LIN {X 0,Y 228.943,Z 711.605,A -85,B 0,C 180,E1 6110.84,E2 6110.84} C_VEL
LIN {X 0,Y 224.559,Z 717.902,A -85,B 0,C 180,E1 6110.576,E2 6110.576} C_VEL
LIN {X 0,Y 211.936,Z 735.349,A -85,B 0,C 180,E1 6108.891,E2 6108.891} C_VEL
LIN {X 0,Y 198.221,Z 751.661,A -85,B 0,C 180,E1 6106.779,E2 6106.779} C_VEL
LIN {X 0,Y 183.955,Z 766.558,A -85,B 0,C 180,E1 6104.16,E2 6104.16} C_VEL
LIN {X 0,Y 168.446,Z 780.857,A -85,B 0,C 180,E1 6100.693,E2 6100.693} C_VEL
LIN {X 0,Y 153.69,Z 792.992,A -85,B 0,C 180,E1 6096.531,E2 6096.531} C_VEL
LIN {X 0,Y 138.441,Z 804.254,A -85,B 0,C 180,E1 6090.912,E2 6090.912} C_VEL
LIN {X 0,Y 124.785,Z 813.422,A -85,B 0,C 180,E1 6084.023,E2 6084.023} C_VEL
LIN {X 0,Y 112.729,Z 821.12,A -85,B 0,C 180,E1 6075.198,E2 6075.198} C_VEL
LIN {X 0,Y 103.673,Z 826.988,A -85,B 0,C 180,E1 6064.681,E2 6064.681} C_VEL
LIN {X 0,Y 98.168,Z 831.113,A -85,B 0,C 180,E1 6052.77,E2 6052.77} C_VEL
LIN {X 0,Y 96.317,Z 833.266,A -85,B 0,C 180,E1 6041.375,E2 6041.375} C_VEL
LIN {X 0,Y 96.353,Z 833.983,A -85,B 0,C 180,E1 6032.974,E2 6032.974} C_VEL
LIN {X 0,Y 96.353,Z 833.978,A -85,B 0,C 180,E1 6027.026,E2 6027.026} C_VEL
LIN {X 0,Y 96.32,Z 833.25,A -85,B 0,C 180,E1 6018.625,E2 6018.625} C_VEL
LIN {X 0,Y 98.345,Z 830.901,A -85,B 0,C 180,E1 6006.641,E2 6006.641} C_VEL
LIN {X 0,Y 104.029,Z 826.718,A -85,B 0,C 180,E1 5994.78,E2 5994.78} C_VEL
LIN {X 0,Y 113.237,Z 820.733,A -85,B 0,C 180,E1 5984.341,E2 5984.341} C_VEL
LIN {X 0,Y 125.437,Z 812.892,A -85,B 0,C 180,E1 5975.582,E2 5975.582} C_VEL
LIN {X 0,Y 139.162,Z 803.604,A -85,B 0,C 180,E1 5968.774,E2 5968.774} C_VEL
LIN {X 0,Y 154.481,Z 792.265,A -85,B 0,C 180,E1 5963.212,E2 5963.212} C_VEL
LIN {X 0,Y 170.131,Z 779.252,A -85,B 0,C 180,E1 5958.885,E2 5958.885} C_VEL
LIN {X 0,Y 184.827,Z 765.494,A -85,B 0,C 180,E1 5955.656,E2 5955.656} C_VEL
LIN {X 0,Y 199.569,Z 749.867,A -85,B 0,C 180,E1 5952.984,E2 5952.984} C_VEL
LIN {X 0,Y 212.851,Z 733.839,A -85,B 0,C 180,E1 5950.966,E2 5950.966} C_VEL
LIN {X 0,Y 225.524,Z 716.172,A -85,B 0,C 180,E1 5949.294,E2 5949.294} C_VEL
LIN {X 0,Y 236.712,Z 697.903,A -85,B 0,C 180,E1 5947.997,E2 5947.997} C_VEL
LIN {X 0,Y 246.77,Z 678.537,A -85,B 0,C 180,E1 5946.946,E2 5946.946} C_VEL
LIN {X 0,Y 255.417,Z 658.457,A -85,B 0,C 180,E1 5946.129,E2 5946.129} C_VEL
LIN {X 0,Y 262.423,Z 638.201,A -85,B 0,C 180,E1 5945.52,E2 5945.52} C_VEL
LIN {X 0,Y 267.944,Z 616.978,A -85,B 0,C 180,E1 5945.047,E2 5945.047} C_VEL
LIN {X 0,Y 271.895,Z 594.865,A -85,B 0,C 180,E1 5944.639,E2 5944.639} C_VEL
LIN {X 0,Y 282.099,Z 508.002,A -85,B 0,C 180,E1 5943.2,E2 5943.2} C_VEL
LIN {X 0,Y 281.259,Z 505.176,A -85,B 0,C 180,E1 5939.389,E2 5939.389} C_VEL
LIN {X 0,Y 281.202,Z 505.463,A -85,B 0,C 180,E1 5936.126,E2 5936.126} C_VEL
LIN {X 0,Y 281.88,Z 508.582,A -85,B 0,C 180,E1 5932.471,E2 5932.471} C_VEL
LIN {X 0,Y 271.081,Z 600.166,A -85,B 0,C 180,E1 5931.031,E2 5931.031} C_VEL
LIN {X 0,Y 266.657,Z 621.932,A -85,B 0,C 180,E1 5930.606,E2 5930.606} C_VEL
LIN {X 0,Y 260.873,Z 642.254,A -85,B 0,C 180,E1 5930.059,E2 5930.059} C_VEL
LIN {X 0,Y 253.227,Z 663.066,A -85,B 0,C 180,E1 5929.305,E2 5929.305} C_VEL
LIN {X 0,Y 244.471,Z 682.335,A -85,B 0,C 180,E1 5928.379,E2 5928.379} C_VEL
LIN {X 0,Y 234.272,Z 700.902,A -85,B 0,C 180,E1 5927.212,E2 5927.212} C_VEL
LIN {X 0,Y 223.26,Z 717.863,A -85,B 0,C 180,E1 5925.826,E2 5925.826} C_VEL
LIN {X 0,Y 210.147,Z 735.251,A -85,B 0,C 180,E1 5923.96,E2 5923.96} C_VEL
LIN {X 0,Y 196.844,Z 750.52,A -85,B 0,C 180,E1 5921.774,E2 5921.774} C_VEL
LIN {X 0,Y 182.156,Z 765.197,A -85,B 0,C 180,E1 5918.924,E2 5918.924} C_VEL
LIN {X 0,Y 167.162,Z 778.201,A -85,B 0,C 180,E1 5915.388,E2 5915.388} C_VEL
LIN {X 0,Y 152.898,Z 789.101,A -85,B 0,C 180,E1 5911.194,E2 5911.194} C_VEL
LIN {X 0,Y 138.176,Z 799.134,A -85,B 0,C 180,E1 5905.578,E2 5905.578} C_VEL
LIN {X 0,Y 124.994,Z 807.232,A -85,B 0,C 180,E1 5898.756,E2 5898.756} C_VEL
LIN {X 0,Y 113.323,Z 813.809,A -85,B 0,C 180,E1 5890.096,E2 5890.096} C_VEL
LIN {X 0,Y 104.467,Z 818.511,A -85,B 0,C 180,E1 5879.847,E2 5879.847} C_VEL
LIN {X 0,Y 98.88,Z 821.593,A -85,B 0,C 180,E1 5868.097,E2 5868.097} C_VEL
LIN {X 0,Y 96.719,Z 823.052,A -85,B 0,C 180,E1 5856.529,E2 5856.529} C_VEL
LIN {X 0,Y 96.52,Z 823.179,A -85,B 0,C 180,E1 5847.031,E2 5847.031} C_VEL
LIN {X 0,Y 97.582,Z 822.439,A -85,B 0,C 180,E1 5836.973,E2 5836.973} C_VEL
LIN {X 0,Y 101.63,Z 820.074,A -85,B 0,C 180,E1 5824.974,E2 5824.974} C_VEL
LIN {X 0,Y 109.093,Z 816.103,A -85,B 0,C 180,E1 5814.087,E2 5814.087} C_VEL
LIN {X 0,Y 119.622,Z 810.413,A -85,B 0,C 180,E1 5804.728,E2 5804.728} C_VEL
LIN {X 0,Y 132.62,Z 802.775,A -85,B 0,C 180,E1 5796.952,E2 5796.952} C_VEL
LIN {X 0,Y 146.033,Z 794.058,A -85,B 0,C 180,E1 5791.149,E2 5791.149} C_VEL
LIN {X 0,Y 161.435,Z 782.868,A -85,B 0,C 180,E1 5786.098,E2 5786.098} C_VEL
LIN {X 0,Y 176.171,Z 770.745,A -85,B 0,C 180,E1 5782.32,E2 5782.32} C_VEL
LIN {X 0,Y 190.669,Z 757.19,A -85,B 0,C 180,E1 5779.286,E2 5779.286} C_VEL
LIN {X 0,Y 204.72,Z 742.023,A -85,B 0,C 180,E1 5776.815,E2 5776.815} C_VEL
LIN {X 0,Y 217.286,Z 726.43,A -85,B 0,C 180,E1 5774.916,E2 5774.916} C_VEL
LIN {X 0,Y 229.6,Z 708.754,A -85,B 0,C 180,E1 5773.278,E2 5773.278} C_VEL
LIN {X 0,Y 240.308,Z 690.764,A -85,B 0,C 180,E1 5772.008,E2 5772.008} C_VEL
LIN {X 0,Y 249.916,Z 671.405,A -85,B 0,C 180,E1 5770.959,E2 5770.959} C_VEL
LIN {X 0,Y 257.672,Z 652.265,A -85,B 0,C 180,E1 5770.173,E2 5770.173} C_VEL
LIN {X 0,Y 264.628,Z 630.575,A -85,B 0,C 180,E1 5769.505,E2 5769.505} C_VEL
LIN {X 0,Y 269.675,Z 609.251,A -85,B 0,C 180,E1 5769.034,E2 5769.034} C_VEL
LIN {X 0,Y 273.096,Z 587.225,A -85,B 0,C 180,E1 5768.661,E2 5768.661} C_VEL
LIN {X 0,Y 282.119,Z 508.77,A -85,B 0,C 180,E1 5767.415,E2 5767.415} C_VEL
LIN {X 0,Y 281.448,Z 505.359,A -85,B 0,C 180,E1 5763.259,E2 5763.259} C_VEL
LIN {X 0,Y 281.564,Z 505.603,A -85,B 0,C 180,E1 5760.204,E2 5760.204} C_VEL
LIN {X 0,Y 282.328,Z 508.47,A -85,B 0,C 180,E1 5756.755,E2 5756.755} C_VEL
LIN {X 0,Y 271.257,Z 601.222,A -85,B 0,C 180,E1 5755.259,E2 5755.259} C_VEL
LIN {X 0,Y 266.713,Z 623.38,A -85,B 0,C 180,E1 5754.832,E2 5754.832} C_VEL
LIN {X 0,Y 260.73,Z 644.157,A -85,B 0,C 180,E1 5754.332,E2 5754.332} C_VEL
LIN {X 0,Y 252.828,Z 665.462,A -85,B 0,C 180,E1 5753.624,E2 5753.624} C_VEL
LIN {X 0,Y 243.909,Z 684.958,A -85,B 0,C 180,E1 5752.749,E2 5752.749} C_VEL
LIN {X 0,Y 233.45,Z 703.978,A -85,B 0,C 180,E1 5751.625,E2 5751.625} C_VEL
LIN {X 0,Y 224.559,Z 717.902,A -85,B 0,C 180,E1 5750.576,E2 5750.576} C_VEL
LIN {X 0,Y 220.012,Z 724.207,A -85,B 0,C 180,E1 5750.279,E2 5750.279} C_VEL
LIN {X 0,Y 206.999,Z 739.459,A -85,B 0,C 180,E1 5750.323,E2 5750.323} C_VEL
LIN {X 0,Y 201.901,Z 745.116,A -85,B 0,C 180,E1 5749.921,E2 5749.921} C_VEL
LIN {X 0,Y 187.314,Z 760.779,A -85,B 0,C 180,E1 5747.635,E2 5747.635} C_VEL
LIN {X 0,Y 172.824,Z 774.387,A -85,B 0,C 180,E1 5744.91,E2 5744.91} C_VEL
LIN {X 0,Y 156.438,Z 787.999,A -85,B 0,C 180,E1 5741.068,E2 5741.068} C_VEL
LIN {X 0,Y 140.822,Z 799.498,A -85,B 0,C 180,E1 5736.333,E2 5736.333} C_VEL
LIN {X 0,Y 125.674,Z 809.548,A -85,B 0,C 180,E1 5730.132,E2 5730.132} C_VEL
LIN {X 0,Y 111.697,Z 817.971,A -85,B 0,C 180,E1 5721.973,E2 5721.973} C_VEL
LIN {X 0,Y 100.404,Z 824.489,A -85,B 0,C 180,E1 5711.85,E2 5711.85} C_VEL
LIN {X 0,Y 92.315,Z 829.427,A -85,B 0,C 180,E1 5699.168,E2 5699.168} C_VEL
LIN {X 0,Y 88.754,Z 832.327,A -85,B 0,C 180,E1 5686.358,E2 5686.358} C_VEL
LIN {X 0,Y 88.313,Z 833.461,A -85,B 0,C 180,E1 5674.936,E2 5674.936} C_VEL
LIN {X 0,Y 88.388,Z 833.582,A -85,B 0,C 180,E1 5668.055,E2 5668.055} C_VEL
LIN {X 0,Y 88.311,Z 832.952,A -85,B 0,C 180,E1 5658.903,E2 5658.903} C_VEL
LIN {X 0,Y 90.258,Z 830.908,A -85,B 0,C 180,E1 5646.498,E2 5646.498} C_VEL
LIN {X 0,Y 96.203,Z 826.924,A -85,B 0,C 180,E1 5633.673,E2 5633.673} C_VEL
LIN {X 0,Y 106.474,Z 820.908,A -85,B 0,C 180,E1 5622.111,E2 5622.111} C_VEL
LIN {X 0,Y 118.725,Z 813.708,A -85,B 0,C 180,E1 5613.517,E2 5613.517} C_VEL
LIN {X 0,Y 133.055,Z 804.664,A -85,B 0,C 180,E1 5606.593,E2 5606.593} C_VEL
LIN {X 0,Y 148.088,Z 794.164,A -85,B 0,C 180,E1 5601.296,E2 5601.296} C_VEL
LIN {X 0,Y 164.141,Z 781.647,A -85,B 0,C 180,E1 5596.995,E2 5596.995} C_VEL
LIN {X 0,Y 179.162,Z 768.454,A -85,B 0,C 180,E1 5593.827,E2 5593.827} C_VEL
LIN {X 0,Y 194.185,Z 753.452,A -85,B 0,C 180,E1 5591.229,E2 5591.229} C_VEL
LIN {X 0,Y 207.964,Z 737.594,A -85,B 0,C 180,E1 5589.235,E2 5589.235} C_VEL
LIN {X 0,Y 220.914,Z 720.48,A -85,B 0,C 180,E1 5587.62,E2 5587.62} C_VEL
LIN {X 0,Y 232.396,Z 702.941,A -85,B 0,C 180,E1 5586.37,E2 5586.37} C_VEL
LIN {X 0,Y 243.011,Z 683.835,A -85,B 0,C 180,E1 5585.334,E2 5585.334} C_VEL
LIN {X 0,Y 251.753,Z 664.803,A -85,B 0,C 180,E1 5584.555,E2 5584.555} C_VEL
LIN {X 0,Y 259.563,Z 643.938,A -85,B 0,C 180,E1 5583.918,E2 5583.918} C_VEL
LIN {X 0,Y 265.684,Z 622.813,A -85,B 0,C 180,E1 5583.45,E2 5583.45} C_VEL
LIN {X 0,Y 270.213,Z 600.861,A -85,B 0,C 180,E1 5583.054,E2 5583.054} C_VEL
LIN {X 0,Y 280.622,Z 514.878,A -85,B 0,C 180,E1 5581.689,E2 5581.689} C_VEL
LIN {X 0,Y 280.248,Z 513.095,A -85,B 0,C 180,E1 5579.182,E2 5579.182} C_VEL
LIN {X 0,Y 280.208,Z 513.353,A -85,B 0,C 180,E1 5576.317,E2 5576.317} C_VEL
LIN {X 0,Y 280.468,Z 515.368,A -85,B 0,C 180,E1 5573.991,E2 5573.991} C_VEL
LIN {X 0,Y 270.229,Z 600.323,A -85,B 0,C 180,E1 5572.716,E2 5572.716} C_VEL
LIN {X 0,Y 265.751,Z 622.044,A -85,B 0,C 180,E1 5572.319,E2 5572.319} C_VEL
LIN {X 0,Y 259.977,Z 642.117,A -85,B 0,C 180,E1 5571.819,E2 5571.819} C_VEL
LIN {X 0,Y 252.47,Z 662.437,A -85,B 0,C 180,E1 5571.14,E2 5571.14} C_VEL
LIN {X 0,Y 244.087,Z 680.892,A -85,B 0,C 180,E1 5570.331,E2 5570.331} C_VEL
LIN {X 0,Y 234.04,Z 699.126,A -85,B 0,C 180,E1 5569.288,E2 5569.288} C_VEL
LIN {X 0,Y 222.222,Z 717.316,A -85,B 0,C 180,E1 5567.932,E2 5567.932} C_VEL
LIN {X 0,Y 209.447,Z 734.138,A -85,B 0,C 180,E1 5566.274,E2 5566.274} C_VEL
LIN {X 0,Y 196.278,Z 749.177,A -85,B 0,C 180,E1 5564.314,E2 5564.314} C_VEL
LIN {X 0,Y 182.04,Z 763.217,A -85,B 0,C 180,E1 5561.838,E2 5561.838} C_VEL
LIN {X 0,Y 167.34,Z 775.94,A -85,B 0,C 180,E1 5558.761,E2 5558.761} C_VEL
LIN {X 0,Y 152.39,Z 787.337,A -85,B 0,C 180,E1 5554.879,E2 5554.879} C_VEL
LIN {X 0,Y 137.245,Z 797.507,A -85,B 0,C 180,E1 5549.822,E2 5549.822} C_VEL
LIN {X 0,Y 122.453,Z 806.219,A -85,B 0,C 180,E1 5543.147,E2 5543.147} C_VEL
LIN {X 0,Y 110.002,Z 812.815,A -85,B 0,C 180,E1 5535.15,E2 5535.15} C_VEL
LIN {X 0,Y 99.13,Z 818.185,A -85,B 0,C 180,E1 5524.39,E2 5524.39} C_VEL
LIN {X 0,Y 92.208,Z 821.597,A -85,B 0,C 180,E1 5512.304,E2 5512.304} C_VEL
LIN {X 0,Y 89.124,Z 823.234,A -85,B 0,C 180,E1 5500.34,E2 5500.34} C_VEL
LIN {X 0,Y 88.502,Z 823.711,A -85,B 0,C 180,E1 5489.353,E2 5489.353} C_VEL
LIN {X 0,Y 89.302,Z 823.135,A -85,B 0,C 180,E1 5478.374,E2 5478.374} C_VEL
LIN {X 0,Y 92.936,Z 821.275,A -85,B 0,C 180,E1 5465.87,E2 5465.87} C_VEL
LIN {X 0,Y 100.36,Z 817.677,A -85,B 0,C 180,E1 5454,E2 5454} C_VEL
LIN {X 0,Y 111.086,Z 812.343,A -85,B 0,C 180,E1 5443.942,E2 5443.942} C_VEL
LIN {X 0,Y 124.421,Z 805.188,A -85,B 0,C 180,E1 5435.745,E2 5435.745} C_VEL
LIN {X 0,Y 138.94,Z 796.519,A -85,B 0,C 180,E1 5429.456,E2 5429.456} C_VEL
LIN {X 0,Y 154.245,Z 786.199,A -85,B 0,C 180,E1 5424.512,E2 5424.512} C_VEL
LIN {X 0,Y 169.828,Z 774.115,A -85,B 0,C 180,E1 5420.597,E2 5420.597} C_VEL
LIN {X 0,Y 184.615,Z 761.006,A -85,B 0,C 180,E1 5417.603,E2 5417.603} C_VEL
LIN {X 0,Y 199.384,Z 745.999,A -85,B 0,C 180,E1 5415.116,E2 5415.116} C_VEL
LIN {X 0,Y 212.601,Z 730.569,A -85,B 0,C 180,E1 5413.222,E2 5413.222} C_VEL
LIN {X 0,Y 225.009,Z 713.713,A -85,B 0,C 180,E1 5411.659,E2 5411.659} C_VEL
LIN {X 0,Y 235.864,Z 696.432,A -85,B 0,C 180,E1 5410.439,E2 5410.439} C_VEL
LIN {X 0,Y 246.247,Z 676.879,A -85,B 0,C 180,E1 5409.374,E2 5409.374} C_VEL
LIN {X 0,Y 254.801,Z 657.342,A -85,B 0,C 180,E1 5408.569,E2 5408.569} C_VEL
LIN {X 0,Y 261.963,Z 636.81,A -85,B 0,C 180,E1 5407.933,E2 5407.933} C_VEL
LIN {X 0,Y 267.47,Z 615.741,A -85,B 0,C 180,E1 5407.456,E2 5407.456} C_VEL
LIN {X 0,Y 271.403,Z 593.852,A -85,B 0,C 180,E1 5407.088,E2 5407.088} C_VEL
LIN {X 0,Y 280.729,Z 515.352,A -85,B 0,C 180,E1 5405.878,E2 5405.878} C_VEL
LIN {X 0,Y 280.444,Z 513.234,A -85,B 0,C 180,E1 5402.657,E2 5402.657} C_VEL
LIN {X 0,Y 280.552,Z 513.477,A -85,B 0,C 180,E1 5400.409,E2 5400.409} C_VEL
LIN {X 0,Y 280.864,Z 515.249,A -85,B 0,C 180,E1 5398.276,E2 5398.276} C_VEL
LIN {X 0,Y 270.432,Z 601.099,A -85,B 0,C 180,E1 5396.948,E2 5396.948} C_VEL
LIN {X 0,Y 265.812,Z 623.347,A -85,B 0,C 180,E1 5396.547,E2 5396.547} C_VEL
LIN {X 0,Y 259.811,Z 643.945,A -85,B 0,C 180,E1 5396.09,E2 5396.09} C_VEL
LIN {X 0,Y 251.756,Z 665.383,A -85,B 0,C 180,E1 5395.434,E2 5395.434} C_VEL
LIN {X 0,Y 243.015,Z 684.289,A -85,B 0,C 180,E1 5394.655,E2 5394.655} C_VEL
LIN {X 0,Y 232.401,Z 703.346,A -85,B 0,C 180,E1 5393.619,E2 5393.619} C_VEL
LIN {X 0,Y 220.919,Z 720.814,A -85,B 0,C 180,E1 5392.369,E2 5392.369} C_VEL
LIN {X 0,Y 207.215,Z 738.779,A -85,B 0,C 180,E1 5390.655,E2 5390.655} C_VEL
LIN {X 0,Y 201.901,Z 745.116,A -85,B 0,C 180,E1 5389.921,E2 5389.921} C_VEL
LIN {X 0,Y 196.629,Z 750.729,A -85,B 0,C 180,E1 5389.468,E2 5389.468} C_VEL
LIN {X 0,Y 181.804,Z 764.258,A -85,B 0,C 180,E1 5389.155,E2 5389.155} C_VEL
LIN {X 0,Y 176.236,Z 769.222,A -85,B 0,C 180,E1 5388.563,E2 5388.563} C_VEL
LIN {X 0,Y 160.13,Z 782.767,A -85,B 0,C 180,E1 5385.42,E2 5385.42} C_VEL
LIN {X 0,Y 143.84,Z 794.82,A -85,B 0,C 180,E1 5381.353,E2 5381.353} C_VEL
LIN {X 0,Y 127.163,Z 805.736,A -85,B 0,C 180,E1 5375.792,E2 5375.792} C_VEL
LIN {X 0,Y 112.21,Z 814.524,A -85,B 0,C 180,E1 5368.803,E2 5368.803} C_VEL
LIN {X 0,Y 98.734,Z 821.792,A -85,B 0,C 180,E1 5359.419,E2 5359.419} C_VEL
LIN {X 0,Y 88.422,Z 827.177,A -85,B 0,C 180,E1 5347.633,E2 5347.633} C_VEL
LIN {X 0,Y 82.171,Z 830.859,A -85,B 0,C 180,E1 5333.674,E2 5333.674} C_VEL
LIN {X 0,Y 80.288,Z 832.717,A -85,B 0,C 180,E1 5320.329,E2 5320.329} C_VEL
LIN {X 0,Y 80.426,Z 833.189,A -85,B 0,C 180,E1 5310.712,E2 5310.712} C_VEL
LIN {X 0,Y 80.269,Z 832.903,A -85,B 0,C 180,E1 5302.125,E2 5302.125} C_VEL
LIN {X 0,Y 81.64,Z 831.213,A -85,B 0,C 180,E1 5288.444,E2 5288.444} C_VEL
LIN {X 0,Y 87.022,Z 827.945,A -85,B 0,C 180,E1 5274.662,E2 5274.662} C_VEL
LIN {X 0,Y 96.492,Z 822.877,A -85,B 0,C 180,E1 5262.635,E2 5262.635} C_VEL
LIN {X 0,Y 108.76,Z 816.303,A -85,B 0,C 180,E1 5253.221,E2 5253.221} C_VEL
LIN {X 0,Y 123.263,Z 808.018,A -85,B 0,C 180,E1 5245.795,E2 5245.795} C_VEL
LIN {X 0,Y 139.357,Z 797.829,A -85,B 0,C 180,E1 5239.97,E2 5239.97} C_VEL
LIN {X 0,Y 155.694,Z 786.056,A -85,B 0,C 180,E1 5235.579,E2 5235.579} C_VEL
LIN {X 0,Y 170.945,Z 773.62,A -85,B 0,C 180,E1 5232.378,E2 5232.378} C_VEL
LIN {X 0,Y 185.715,Z 760.038,A -85,B 0,C 180,E1 5229.865,E2 5229.865} C_VEL
LIN {X 0,Y 200.792,Z 744.156,A -85,B 0,C 180,E1 5227.733,E2 5227.733} C_VEL
LIN {X 0,Y 214.187,Z 727.761,A -85,B 0,C 180,E1 5226.127,E2 5226.127} C_VEL
LIN {X 0,Y 226.921,Z 709.717,A -85,B 0,C 180,E1 5224.802,E2 5224.802} C_VEL
LIN {X 0,Y 237.98,Z 691.361,A -85,B 0,C 180,E1 5223.789,E2 5223.789} C_VEL
LIN {X 0,Y 247.792,Z 671.982,A -85,B 0,C 180,E1 5222.974,E2 5222.974} C_VEL
LIN {X 0,Y 256.17,Z 651.514,A -85,B 0,C 180,E1 5222.337,E2 5222.337} C_VEL
LIN {X 0,Y 262.969,Z 630.411,A -85,B 0,C 180,E1 5221.863,E2 5221.863} C_VEL
LIN {X 0,Y 268.333,Z 607.61,A -85,B 0,C 180,E1 5221.467,E2 5221.467} C_VEL
LIN {X 0,Y 271.894,Z 583.958,A -85,B 0,C 180,E1 5221.1,E2 5221.1} C_VEL
LIN {X 0,Y 279.349,Z 521.673,A -85,B 0,C 180,E1 5220.153,E2 5220.153} C_VEL
LIN {X 0,Y 279.221,Z 520.995,A -85,B 0,C 180,E1 5218.768,E2 5218.768} C_VEL
LIN {X 0,Y 279.217,Z 521.278,A -85,B 0,C 180,E1 5216.467,E2 5216.467} C_VEL
LIN {X 0,Y 279.239,Z 522.27,A -85,B 0,C 180,E1 5215.53,E2 5215.53} C_VEL
LIN {X 0,Y 269.581,Z 600.652,A -85,B 0,C 180,E1 5214.408,E2 5214.408} C_VEL
LIN {X 0,Y 265.02,Z 622.436,A -85,B 0,C 180,E1 5214.038,E2 5214.038} C_VEL
LIN {X 0,Y 259.173,Z 642.455,A -85,B 0,C 180,E1 5213.576,E2 5213.576} C_VEL
LIN {X 0,Y 251.366,Z 663.216,A -85,B 0,C 180,E1 5212.934,E2 5212.934} C_VEL
LIN {X 0,Y 242.722,Z 681.885,A -85,B 0,C 180,E1 5212.172,E2 5212.172} C_VEL
LIN {X 0,Y 231.736,Z 701.355,A -85,B 0,C 180,E1 5211.125,E2 5211.125} C_VEL
LIN {X 0,Y 219.887,Z 719.001,A -85,B 0,C 180,E1 5209.876,E2 5209.876} C_VEL
LIN {X 0,Y 206.289,Z 736.307,A -85,B 0,C 180,E1 5208.249,E2 5208.249} C_VEL
LIN {X 0,Y 192.419,Z 751.52,A -85,B 0,C 180,E1 5206.329,E2 5206.329} C_VEL
LIN {X 0,Y 177.894,Z 765.368,A -85,B 0,C 180,E1 5203.963,E2 5203.963} C_VEL
LIN {X 0,Y 162.838,Z 777.788,A -85,B 0,C 180,E1 5201.008,E2 5201.008} C_VEL
LIN {X 0,Y 146.622,Z 789.48,A -85,B 0,C 180,E1 5197.011,E2 5197.011} C_VEL
LIN {X 0,Y 131.261,Z 799.17,A -85,B 0,C 180,E1 5192.078,E2 5192.078} C_VEL
LIN {X 0,Y 116.349,Z 807.457,A -85,B 0,C 180,E1 5185.585,E2 5185.585} C_VEL
LIN {X 0,Y 102.63,Z 814.144,A -85,B 0,C 180,E1 5176.941,E2 5176.941} C_VEL
LIN {X 0,Y 91.658,Z 819.03,A -85,B 0,C 180,E1 5166.09,E2 5166.09} C_VEL
LIN {X 0,Y 84.017,Z 822.363,A -85,B 0,C 180,E1 5152.384,E2 5152.384} C_VEL
LIN {X 0,Y 80.974,Z 823.873,A -85,B 0,C 180,E1 5139.237,E2 5139.237} C_VEL
LIN {X 0,Y 80.526,Z 824.117,A -85,B 0,C 180,E1 5127.865,E2 5127.865} C_VEL
LIN {X 0,Y 81.711,Z 823.463,A -85,B 0,C 180,E1 5115.834,E2 5115.834} C_VEL
LIN {X 0,Y 86.574,Z 821.28,A -85,B 0,C 180,E1 5101.738,E2 5101.738} C_VEL
LIN {X 0,Y 95.41,Z 817.497,A -85,B 0,C 180,E1 5089.48,E2 5089.48} C_VEL
LIN {X 0,Y 107.519,Z 811.925,A -85,B 0,C 180,E1 5079.482,E2 5079.482} C_VEL
LIN {X 0,Y 121.324,Z 804.86,A -85,B 0,C 180,E1 5071.916,E2 5071.916} C_VEL
LIN {X 0,Y 136.736,Z 795.977,A -85,B 0,C 180,E1 5065.922,E2 5065.922} C_VEL
LIN {X 0,Y 152.446,Z 785.662,A -85,B 0,C 180,E1 5061.359,E2 5061.359} C_VEL
LIN {X 0,Y 168.042,Z 773.9,A -85,B 0,C 180,E1 5057.827,E2 5057.827} C_VEL
LIN {X 0,Y 183.245,Z 760.66,A -85,B 0,C 180,E1 5055.037,E2 5055.037} C_VEL
LIN {X 0,Y 197.884,Z 746.026,A -85,B 0,C 180,E1 5052.8,E2 5052.8} C_VEL
LIN {X 0,Y 211.486,Z 730.369,A -85,B 0,C 180,E1 5051.028,E2 5051.028} C_VEL
LIN {X 0,Y 224.093,Z 713.486,A -85,B 0,C 180,E1 5049.589,E2 5049.589} C_VEL
LIN {X 0,Y 235.502,Z 695.444,A -85,B 0,C 180,E1 5048.426,E2 5048.426} C_VEL
LIN {X 0,Y 245.616,Z 676.461,A -85,B 0,C 180,E1 5047.485,E2 5047.485} C_VEL
LIN {X 0,Y 254.171,Z 657.038,A -85,B 0,C 180,E1 5046.755,E2 5046.755} C_VEL
LIN {X 0,Y 261.469,Z 636.272,A -85,B 0,C 180,E1 5046.166,E2 5046.166} C_VEL
LIN {X 0,Y 267.092,Z 614.729,A -85,B 0,C 180,E1 5045.723,E2 5045.723} C_VEL
LIN {X 0,Y 270.917,Z 593.231,A -85,B 0,C 180,E1 5045.389,E2 5045.389} C_VEL
LIN {X 0,Y 279.51,Z 522.254,A -85,B 0,C 180,E1 5044.36,E2 5044.36} C_VEL
LIN {X 0,Y 279.455,Z 521.163,A -85,B 0,C 180,E1 5042.461,E2 5042.461} C_VEL
LIN {X 0,Y 279.556,Z 521.508,A -85,B 0,C 180,E1 5040.41,E2 5040.41} C_VEL
LIN {X 0,Y 279.581,Z 522.193,A -85,B 0,C 180,E1 5039.808,E2 5039.808} C_VEL
LIN {X 0,Y 269.842,Z 600.976,A -85,B 0,C 180,E1 5038.645,E2 5038.645} C_VEL
LIN {X 0,Y 265.194,Z 623.129,A -85,B 0,C 180,E1 5038.274,E2 5038.274} C_VEL
LIN {X 0,Y 259.137,Z 643.734,A -85,B 0,C 180,E1 5037.859,E2 5037.859} C_VEL
LIN {X 0,Y 251.24,Z 664.606,A -85,B 0,C 180,E1 5037.281,E2 5037.281} C_VEL
LIN {X 0,Y 242.392,Z 683.62,A -85,B 0,C 180,E1 5036.573,E2 5036.573} C_VEL
LIN {X 0,Y 231.635,Z 702.715,A -85,B 0,C 180,E1 5035.628,E2 5035.628} C_VEL
LIN {X 0,Y 219.981,Z 720.24,A -85,B 0,C 180,E1 5034.486,E2 5034.486} C_VEL
LIN {X 0,Y 206.201,Z 738.053,A -85,B 0,C 180,E1 5032.931,E2 5032.931} C_VEL
LIN {X 0,Y 192.282,Z 753.643,A -85,B 0,C 180,E1 5031.102,E2 5031.102} C_VEL
LIN {X 0,Y 177.372,Z 768.155,A -85,B 0,C 180,E1 5028.76,E2 5028.76} C_VEL
LIN {X 0,Y 176.236,Z 769.222,A -85,B 0,C 180,E1 5028.563,E2 5028.563} C_VEL
LIN {X 0,Y 170.514,Z 774.076,A -85,B 0,C 180,E1 5027.902,E2 5027.902} C_VEL
LIN {X 0,Y 154.154,Z 785.624,A -85,B 0,C 180,E1 5027.075,E2 5027.075} C_VEL
LIN {X 0,Y 148.092,Z 789.773,A -85,B 0,C 180,E1 5026.169,E2 5026.169} C_VEL
LIN {X 0,Y 131.558,Z 800.689,A -85,B 0,C 180,E1 5021.803,E2 5021.803} C_VEL
LIN {X 0,Y 114.28,Z 810.736,A -85,B 0,C 180,E1 5015.49,E2 5015.49} C_VEL
LIN {X 0,Y 99.483,Z 818.433,A -85,B 0,C 180,E1 5007.589,E2 5007.589} C_VEL
LIN {X 0,Y 86.509,Z 824.644,A -85,B 0,C 180,E1 4996.729,E2 4996.729} C_VEL
LIN {X 0,Y 77.274,Z 829.029,A -85,B 0,C 180,E1 4982.917,E2 4982.917} C_VEL
LIN {X 0,Y 72.755,Z 831.739,A -85,B 0,C 180,E1 4966.774,E2 4966.774} C_VEL
LIN {X 0,Y 72.336,Z 832.607,A -85,B 0,C 180,E1 4954.757,E2 4954.757} C_VEL
LIN {X 0,Y 72.397,Z 832.684,A -85,B 0,C 180,E1 4947.625,E2 4947.625} C_VEL
LIN {X 0,Y 72.45,Z 832.041,A -85,B 0,C 180,E1 4936.432,E2 4936.432} C_VEL
LIN {X 0,Y 75.472,Z 829.986,A -85,B 0,C 180,E1 4921.516,E2 4921.516} C_VEL
LIN {X 0,Y 83.439,Z 825.993,A -85,B 0,C 180,E1 4906.92,E2 4906.92} C_VEL
LIN {X 0,Y 96.109,Z 819.968,A -85,B 0,C 180,E1 4894.73,E2 4894.73} C_VEL
LIN {X 0,Y 110.396,Z 812.76,A -85,B 0,C 180,E1 4886.283,E2 4886.283} C_VEL
LIN {X 0,Y 126.476,Z 803.717,A -85,B 0,C 180,E1 4879.826,E2 4879.826} C_VEL
LIN {X 0,Y 142.887,Z 793.202,A -85,B 0,C 180,E1 4875.065,E2 4875.065} C_VEL
LIN {X 0,Y 159.16,Z 781.385,A -85,B 0,C 180,E1 4871.484,E2 4871.484} C_VEL
LIN {X 0,Y 175,Z 768.306,A -85,B 0,C 180,E1 4868.734,E2 4868.734} C_VEL
LIN {X 0,Y 190.216,Z 753.845,A -85,B 0,C 180,E1 4866.567,E2 4866.567} C_VEL
LIN {X 0,Y 204.699,Z 737.987,A -85,B 0,C 180,E1 4864.852,E2 4864.852} C_VEL
LIN {X 0,Y 218.362,Z 720.675,A -85,B 0,C 180,E1 4863.464,E2 4863.464} C_VEL
LIN {X 0,Y 230.167,Z 703.304,A -85,B 0,C 180,E1 4862.424,E2 4862.424} C_VEL
LIN {X 0,Y 241.049,Z 684.298,A -85,B 0,C 180,E1 4861.564,E2 4861.564} C_VEL
LIN {X 0,Y 250.095,Z 665.261,A -85,B 0,C 180,E1 4860.916,E2 4860.916} C_VEL
LIN {X 0,Y 258.212,Z 644.223,A -85,B 0,C 180,E1 4860.385,E2 4860.385} C_VEL
LIN {X 0,Y 264.456,Z 623.316,A -85,B 0,C 180,E1 4860.002,E2 4860.002} C_VEL
LIN {X 0,Y 269.178,Z 601.085,A -85,B 0,C 180,E1 4859.658,E2 4859.658} C_VEL
LIN {X 0,Y 277.839,Z 532.135,A -85,B 0,C 180,E1 4858.689,E2 4858.689} C_VEL
LIN {X 0,Y 278.228,Z 528.921,A -85,B 0,C 180,E1 4858.613,E2 4858.613} C_VEL
LIN {X 0,Y 278.198,Z 529.135,A -85,B 0,C 180,E1 4857.082,E2 4857.082} C_VEL
LIN {X 0,Y 269.2,Z 600.807,A -85,B 0,C 180,E1 4856.109,E2 4856.109} C_VEL
LIN {X 0,Y 264.555,Z 622.721,A -85,B 0,C 180,E1 4855.766,E2 4855.766} C_VEL
LIN {X 0,Y 258.613,Z 642.792,A -85,B 0,C 180,E1 4855.343,E2 4855.343} C_VEL
LIN {X 0,Y 250.678,Z 663.613,A -85,B 0,C 180,E1 4854.754,E2 4854.754} C_VEL
LIN {X 0,Y 241.764,Z 682.552,A -85,B 0,C 180,E1 4854.045,E2 4854.045} C_VEL
LIN {X 0,Y 231.12,Z 701.181,A -85,B 0,C 180,E1 4853.13,E2 4853.13} C_VEL
LIN {X 0,Y 219.368,Z 718.54,A -85,B 0,C 180,E1 4852.019,E2 4852.019} C_VEL
LIN {X 0,Y 205.754,Z 735.739,A -85,B 0,C 180,E1 4850.556,E2 4850.556} C_VEL
LIN {X 0,Y 191.615,Z 751.107,A -85,B 0,C 180,E1 4848.803,E2 4848.803} C_VEL
LIN {X 0,Y 176.181,Z 765.55,A -85,B 0,C 180,E1 4846.544,E2 4846.544} C_VEL
LIN {X 0,Y 160.392,Z 778.266,A -85,B 0,C 180,E1 4843.737,E2 4843.737} C_VEL
LIN {X 0,Y 143.655,Z 789.949,A -85,B 0,C 180,E1 4839.983,E2 4839.983} C_VEL
LIN {X 0,Y 126.849,Z 800.077,A -85,B 0,C 180,E1 4835.017,E2 4835.017} C_VEL
LIN {X 0,Y 111.216,Z 808.264,A -85,B 0,C 180,E1 4828.654,E2 4828.654} C_VEL
LIN {X 0,Y 96.634,Z 814.893,A -85,B 0,C 180,E1 4819.964,E2 4819.964} C_VEL
LIN {X 0,Y 84.76,Z 819.681,A -85,B 0,C 180,E1 4808.696,E2 4808.696} C_VEL
LIN {X 0,Y 76.343,Z 822.921,A -85,B 0,C 180,E1 4793.953,E2 4793.953} C_VEL
LIN {X 0,Y 72.987,Z 824.377,A -85,B 0,C 180,E1 4779.461,E2 4779.461} C_VEL
LIN {X 0,Y 72.559,Z 824.544,A -85,B 0,C 180,E1 4766.84,E2 4766.84} C_VEL
LIN {X 0,Y 74.115,Z 823.851,A -85,B 0,C 180,E1 4753.543,E2 4753.543} C_VEL
LIN {X 0,Y 79.953,Z 821.571,A -85,B 0,C 180,E1 4738.255,E2 4738.255} C_VEL
LIN {X 0,Y 89.962,Z 817.708,A -85,B 0,C 180,E1 4725.559,E2 4725.559} C_VEL
LIN {X 0,Y 103.423,Z 812.014,A -85,B 0,C 180,E1 4715.456,E2 4715.456} C_VEL
LIN {X 0,Y 118.795,Z 804.533,A -85,B 0,C 180,E1 4707.905,E2 4707.905} C_VEL
LIN {X 0,Y 135.07,Z 795.435,A -85,B 0,C 180,E1 4702.288,E2 4702.288} C_VEL
LIN {X 0,Y 152.327,Z 784.266,A -85,B 0,C 180,E1 4697.873,E2 4697.873} C_VEL
LIN {X 0,Y 168.471,Z 772.182,A -85,B 0,C 180,E1 4694.678,E2 4694.678} C_VEL
LIN {X 0,Y 184.105,Z 758.656,A -85,B 0,C 180,E1 4692.167,E2 4692.167} C_VEL
LIN {X 0,Y 199.086,Z 743.538,A -85,B 0,C 180,E1 4690.157,E2 4690.157} C_VEL
LIN {X 0,Y 212.846,Z 727.445,A -85,B 0,C 180,E1 4688.58,E2 4688.58} C_VEL
LIN {X 0,Y 225.783,Z 709.785,A -85,B 0,C 180,E1 4687.281,E2 4687.281} C_VEL
LIN {X 0,Y 236.885,Z 692,A -85,B 0,C 180,E1 4686.289,E2 4686.289} C_VEL
LIN {X 0,Y 247.075,Z 672.32,A -85,B 0,C 180,E1 4685.45,E2 4685.45} C_VEL
LIN {X 0,Y 255.138,Z 653.236,A -85,B 0,C 180,E1 4684.834,E2 4684.834} C_VEL
LIN {X 0,Y 262.446,Z 631.367,A -85,B 0,C 180,E1 4684.304,E2 4684.304} C_VEL
LIN {X 0,Y 267.679,Z 610.222,A -85,B 0,C 180,E1 4683.935,E2 4683.935} C_VEL
LIN {X 0,Y 271.309,Z 588.121,A -85,B 0,C 180,E1 4683.624,E2 4683.624} C_VEL
LIN {X 0,Y 278.477,Z 529.125,A -85,B 0,C 180,E1 4682.779,E2 4682.779} C_VEL
LIN {X 0,Y 278.483,Z 529.264,A -85,B 0,C 180,E1 4681.352,E2 4681.352} C_VEL
LIN {X 0,Y 269.459,Z 601.031,A -85,B 0,C 180,E1 4680.345,E2 4680.345} C_VEL
LIN {X 0,Y 264.73,Z 623.284,A -85,B 0,C 180,E1 4680.002,E2 4680.002} C_VEL
LIN {X 0,Y 258.462,Z 644.269,A -85,B 0,C 180,E1 4679.62,E2 4679.62} C_VEL
LIN {X 0,Y 250.27,Z 665.472,A -85,B 0,C 180,E1 4679.085,E2 4679.085} C_VEL
LIN {X 0,Y 241.05,Z 684.775,A -85,B 0,C 180,E1 4678.425,E2 4678.425} C_VEL
LIN {X 0,Y 230.169,Z 703.73,A -85,B 0,C 180,E1 4677.563,E2 4677.563} C_VEL
LIN {X 0,Y 218.364,Z 721.026,A -85,B 0,C 180,E1 4676.525,E2 4676.525} C_VEL
LIN {X 0,Y 204.702,Z 738.275,A -85,B 0,C 180,E1 4675.137,E2 4675.137} C_VEL
LIN {X 0,Y 190.22,Z 754.081,A -85,B 0,C 180,E1 4673.423,E2 4673.423} C_VEL
LIN {X 0,Y 175.004,Z 768.519,A -85,B 0,C 180,E1 4671.257,E2 4671.257} C_VEL
LIN {X 0,Y 159.165,Z 781.56,A -85,B 0,C 180,E1 4668.508,E2 4668.508} C_VEL
LIN {X 0,Y 148.092,Z 789.773,A -85,B 0,C 180,E1 4666.169,E2 4666.169} C_VEL
LIN {X 0,Y 141.968,Z 793.804,A -85,B 0,C 180,E1 4665.159,E2 4665.159} C_VEL
LIN {X 0,Y 124.578,Z 803.209,A -85,B 0,C 180,E1 4663.45,E2 4663.45} C_VEL
LIN {X 0,Y 118.265,Z 806.465,A -85,B 0,C 180,E1 4662.008,E2 4662.008} C_VEL
LIN {X 0,Y 101.386,Z 815.076,A -85,B 0,C 180,E1 4655.13,E2 4655.13} C_VEL
LIN {X 0,Y 86.107,Z 822.004,A -85,B 0,C 180,E1 4645.529,E2 4645.529} C_VEL
LIN {X 0,Y 73.98,Z 827.141,A -85,B 0,C 180,E1 4632.512,E2 4632.512} C_VEL
LIN {X 0,Y 66.426,Z 830.45,A -85,B 0,C 180,E1 4615.881,E2 4615.881} C_VEL
LIN {X 0,Y 64.286,Z 832.033,A -85,B 0,C 180,E1 4598.947,E2 4598.947} C_VEL
LIN {X 0,Y 64.442,Z 832.287,A -85,B 0,C 180,E1 4589.111,E2 4589.111} C_VEL
LIN {X 0,Y 64.385,Z 831.822,A -85,B 0,C 180,E1 4577.443,E2 4577.443} C_VEL
LIN {X 0,Y 67.451,Z 829.909,A -85,B 0,C 180,E1 4560.715,E2 4560.715} C_VEL
LIN {X 0,Y 76.511,Z 825.974,A -85,B 0,C 180,E1 4544.05,E2 4544.05} C_VEL
LIN {X 0,Y 89.504,Z 820.463,A -85,B 0,C 180,E1 4531.9,E2 4531.9} C_VEL
LIN {X 0,Y 105.351,Z 813.126,A -85,B 0,C 180,E1 4522.99,E2 4522.99} C_VEL
LIN {X 0,Y 123.023,Z 803.721,A -85,B 0,C 180,E1 4516.462,E2 4516.462} C_VEL
LIN {X 0,Y 140.039,Z 793.315,A -85,B 0,C 180,E1 4512.003,E2 4512.003} C_VEL
LIN {X 0,Y 157.718,Z 780.897,A -85,B 0,C 180,E1 4508.53,E2 4508.53} C_VEL
LIN {X 0,Y 173.936,Z 767.802,A -85,B 0,C 180,E1 4506.038,E2 4506.038} C_VEL
LIN {X 0,Y 189.45,Z 753.333,A -85,B 0,C 180,E1 4504.088,E2 4504.088} C_VEL
LIN {X 0,Y 204.168,Z 737.447,A -85,B 0,C 180,E1 4502.552,E2 4502.552} C_VEL
LIN {X 0,Y 218.02,Z 720.094,A -85,B 0,C 180,E1 4501.313,E2 4501.313} C_VEL
LIN {X 0,Y 229.966,Z 702.662,A -85,B 0,C 180,E1 4500.39,E2 4500.39} C_VEL
LIN {X 0,Y 240.964,Z 683.617,A -85,B 0,C 180,E1 4499.627,E2 4499.627} C_VEL
LIN {X 0,Y 249.991,Z 664.709,A -85,B 0,C 180,E1 4499.061,E2 4499.061} C_VEL
LIN {X 0,Y 258.033,Z 643.992,A -85,B 0,C 180,E1 4498.601,E2 4498.601} C_VEL
LIN {X 0,Y 264.348,Z 622.961,A -85,B 0,C 180,E1 4498.26,E2 4498.26} C_VEL
LIN {X 0,Y 269.096,Z 600.749,A -85,B 0,C 180,E1 4497.946,E2 4497.946} C_VEL
LIN {X 0,Y 269.768,Z 596.228,A -85,B 0,C 180,E1 4497.874,E2 4497.874} C_VEL
LIN {X 0,Y 265.412,Z 618.489,A -85,B 0,C 180,E1 4497.571,E2 4497.571} C_VEL
LIN {X 0,Y 259.517,Z 639.518,A -85,B 0,C 180,E1 4497.196,E2 4497.196} C_VEL
LIN {X 0,Y 252.369,Z 659.102,A -85,B 0,C 180,E1 4496.725,E2 4496.725} C_VEL
LIN {X 0,Y 243.518,Z 678.392,A -85,B 0,C 180,E1 4496.114,E2 4496.114} C_VEL
LIN {X 0,Y 232.743,Z 697.799,A -85,B 0,C 180,E1 4495.302,E2 4495.302} C_VEL
LIN {X 0,Y 221.043,Z 715.518,A -85,B 0,C 180,E1 4494.333,E2 4494.333} C_VEL
LIN {X 0,Y 207.726,Z 732.7,A -85,B 0,C 180,E1 4493.088,E2 4493.088} C_VEL
LIN {X 0,Y 193.078,Z 748.729,A -85,B 0,C 180,E1 4491.52,E2 4491.52} C_VEL
LIN {X 0,Y 177.892,Z 763.033,A -85,B 0,C 180,E1 4489.602,E2 4489.602} C_VEL
LIN {X 0,Y 161.086,Z 776.683,A -85,B 0,C 180,E1 4487.025,E2 4487.025} C_VEL
LIN {X 0,Y 144.671,Z 788.175,A -85,B 0,C 180,E1 4483.871,E2 4483.871} C_VEL
LIN {X 0,Y 127.066,Z 798.736,A -85,B 0,C 180,E1 4479.449,E2 4479.449} C_VEL
LIN {X 0,Y 110.027,Z 807.393,A -85,B 0,C 180,E1 4473.558,E2 4473.558} C_VEL
LIN {X 0,Y 94.431,Z 814.189,A -85,B 0,C 180,E1 4465.676,E2 4465.676} C_VEL
LIN {X 0,Y 80.261,Z 819.552,A -85,B 0,C 180,E1 4454.235,E2 4454.235} C_VEL
LIN {X 0,Y 70.408,Z 822.955,A -85,B 0,C 180,E1 4439.803,E2 4439.803} C_VEL
LIN {X 0,Y 65.59,Z 824.585,A -85,B 0,C 180,E1 4424.117,E2 4424.117} C_VEL
LIN {X 0,Y 64.54,Z 825.056,A -85,B 0,C 180,E1 4409.112,E2 4409.112} C_VEL
LIN {X 0,Y 65.887,Z 824.486,A -85,B 0,C 180,E1 4394.148,E2 4394.148} C_VEL
LIN {X 0,Y 71.511,Z 822.634,A -85,B 0,C 180,E1 4377.907,E2 4377.907} C_VEL
LIN {X 0,Y 81.949,Z 819.035,A -85,B 0,C 180,E1 4363.959,E2 4363.959} C_VEL
LIN {X 0,Y 95.812,Z 813.704,A -85,B 0,C 180,E1 4353.402,E2 4353.402} C_VEL
LIN {X 0,Y 111.958,Z 806.555,A -85,B 0,C 180,E1 4345.581,E2 4345.581} C_VEL
LIN {X 0,Y 127.873,Z 798.404,A -85,B 0,C 180,E1 4340.237,E2 4340.237} C_VEL
LIN {X 0,Y 144.682,Z 788.318,A -85,B 0,C 180,E1 4336.048,E2 4336.048} C_VEL
LIN {X 0,Y 161.04,Z 776.898,A -85,B 0,C 180,E1 4332.904,E2 4332.904} C_VEL
LIN {X 0,Y 177.851,Z 763.294,A -85,B 0,C 180,E1 4330.326,E2 4330.326} C_VEL
LIN {X 0,Y 193.042,Z 749.039,A -85,B 0,C 180,E1 4328.408,E2 4328.408} C_VEL
LIN {X 0,Y 207.452,Z 733.321,A -85,B 0,C 180,E1 4326.863,E2 4326.863} C_VEL
LIN {X 0,Y 220.529,Z 716.582,A -85,B 0,C 180,E1 4325.636,E2 4325.636} C_VEL
LIN {X 0,Y 232.718,Z 698.282,A -85,B 0,C 180,E1 4324.625,E2 4324.625} C_VEL
LIN {X 0,Y 243.497,Z 678.987,A -85,B 0,C 180,E1 4323.812,E2 4323.812} C_VEL
LIN {X 0,Y 252.351,Z 659.838,A -85,B 0,C 180,E1 4323.202,E2 4323.202} C_VEL
LIN {X 0,Y 259.995,Z 638.912,A -85,B 0,C 180,E1 4322.7,E2 4322.7} C_VEL
LIN {X 0,Y 265.831,Z 617.891,A -85,B 0,C 180,E1 4322.329,E2 4322.329} C_VEL
LIN {X 0,Y 269.556,Z 599.574,A -85,B 0,C 180,E1 4322.07,E2 4322.07} C_VEL
LIN {X 0,Y 265.044,Z 621.204,A -85,B 0,C 180,E1 4321.767,E2 4321.767} C_VEL
LIN {X 0,Y 258.786,Z 642.562,A -85,B 0,C 180,E1 4321.427,E2 4321.427} C_VEL
LIN {X 0,Y 250.994,Z 663.047,A -85,B 0,C 180,E1 4320.986,E2 4320.986} C_VEL
LIN {X 0,Y 241.966,Z 682.258,A -85,B 0,C 180,E1 4320.426,E2 4320.426} C_VEL
LIN {X 0,Y 230.964,Z 701.454,A -85,B 0,C 180,E1 4319.673,E2 4319.673} C_VEL
LIN {X 0,Y 219.014,Z 719.096,A -85,B 0,C 180,E1 4318.758,E2 4318.758} C_VEL
LIN {X 0,Y 205.155,Z 736.612,A -85,B 0,C 180,E1 4317.532,E2 4317.532} C_VEL
LIN {X 0,Y 190.429,Z 752.629,A -85,B 0,C 180,E1 4316.012,E2 4316.012} C_VEL
LIN {X 0,Y 173.939,Z 768.02,A -85,B 0,C 180,E1 4313.952,E2 4313.952} C_VEL
LIN {X 0,Y 157.722,Z 781.074,A -85,B 0,C 180,E1 4311.461,E2 4311.461} C_VEL
LIN {X 0,Y 140.042,Z 793.46,A -85,B 0,C 180,E1 4307.989,E2 4307.989} C_VEL
LIN {X 0,Y 122.692,Z 804.021,A -85,B 0,C 180,E1 4303.428,E2 4303.428} C_VEL
LIN {X 0,Y 118.265,Z 806.465,A -85,B 0,C 180,E1 4302.008,E2 4302.008} C_VEL
LIN {X 0,Y 111.957,Z 809.622,A -85,B 0,C 180,E1 4300.377,E2 4300.377} C_VEL
LIN {X 0,Y 93.192,Z 817.04,A -85,B 0,C 180,E1 4296.612,E2 4296.612} C_VEL
LIN {X 0,Y 87.933,Z 819.011,A -85,B 0,C 180,E1 4294.371,E2 4294.371} C_VEL
LIN {X 0,Y 72.842,Z 824.891,A -85,B 0,C 180,E1 4282.76,E2 4282.76} C_VEL
LIN {X 0,Y 61.899,Z 828.964,A -85,B 0,C 180,E1 4266.701,E2 4266.701} C_VEL
LIN {X 0,Y 56.76,Z 831.145,A -85,B 0,C 180,E1 4247.425,E2 4247.425} C_VEL
LIN {X 0,Y 56.421,Z 831.817,A -85,B 0,C 180,E1 4232.031,E2 4232.031} C_VEL
LIN {X 0,Y 56.309,Z 831.668,A -85,B 0,C 180,E1 4222.86,E2 4222.86} C_VEL
LIN {X 0,Y 58.117,Z 830.468,A -85,B 0,C 180,E1 4204.526,E2 4204.526} C_VEL
LIN {X 0,Y 65.483,Z 827.535,A -85,B 0,C 180,E1 4186.6,E2 4186.6} C_VEL
LIN {X 0,Y 78.828,Z 822.562,A -85,B 0,C 180,E1 4171.81,E2 4171.81} C_VEL
LIN {X 0,Y 94.868,Z 816.006,A -85,B 0,C 180,E1 4161.96,E2 4161.96} C_VEL
LIN {X 0,Y 111.949,Z 807.999,A -85,B 0,C 180,E1 4155.299,E2 4155.299} C_VEL
LIN {X 0,Y 130.123,Z 798.008,A -85,B 0,C 180,E1 4150.416,E2 4150.416} C_VEL
LIN {X 0,Y 148.048,Z 786.569,A -85,B 0,C 180,E1 4146.902,E2 4146.902} C_VEL
LIN {X 0,Y 165.437,Z 773.715,A -85,B 0,C 180,E1 4144.299,E2 4144.299} C_VEL
LIN {X 0,Y 181.13,Z 760.372,A -85,B 0,C 180,E1 4142.417,E2 4142.417} C_VEL
LIN {X 0,Y 196.709,Z 744.94,A -85,B 0,C 180,E1 4140.873,E2 4140.873} C_VEL
LIN {X 0,Y 210.967,Z 728.563,A -85,B 0,C 180,E1 4139.683,E2 4139.683} C_VEL
LIN {X 0,Y 224.354,Z 710.618,A -85,B 0,C 180,E1 4138.723,E2 4138.723} C_VEL
LIN {X 0,Y 236.106,Z 692.053,A -85,B 0,C 180,E1 4137.985,E2 4137.985} C_VEL
LIN {X 0,Y 239.703,Z 685.557,A -85,B 0,C 180,E1 4137.774,E2 4137.774} C_VEL
LIN {X 0,Y 228.77,Z 703.987,A -85,B 0,C 180,E1 4137.019,E2 4137.019} C_VEL
LIN {X 0,Y 216.466,Z 721.363,A -85,B 0,C 180,E1 4136.095,E2 4136.095} C_VEL
LIN {X 0,Y 202.761,Z 737.889,A -85,B 0,C 180,E1 4134.925,E2 4134.925} C_VEL
LIN {X 0,Y 187.215,Z 753.93,A -85,B 0,C 180,E1 4133.385,E2 4133.385} C_VEL
LIN {X 0,Y 171.826,Z 767.607,A -85,B 0,C 180,E1 4131.573,E2 4131.573} C_VEL
LIN {X 0,Y 154.757,Z 780.592,A -85,B 0,C 180,E1 4129.118,E2 4129.118} C_VEL
LIN {X 0,Y 138.031,Z 791.442,A -85,B 0,C 180,E1 4126.08,E2 4126.08} C_VEL
LIN {X 0,Y 120.015,Z 801.444,A -85,B 0,C 180,E1 4121.753,E2 4121.753} C_VEL
LIN {X 0,Y 102.876,Z 809.519,A -85,B 0,C 180,E1 4116.003,E2 4116.003} C_VEL
LIN {X 0,Y 86.35,Z 816.097,A -85,B 0,C 180,E1 4107.699,E2 4107.699} C_VEL
LIN {X 0,Y 72.229,Z 820.788,A -85,B 0,C 180,E1 4096.039,E2 4096.039} C_VEL
LIN {X 0,Y 61.946,Z 823.828,A -85,B 0,C 180,E1 4080.023,E2 4080.023} C_VEL
LIN {X 0,Y 57.197,Z 825.286,A -85,B 0,C 180,E1 4061.77,E2 4061.77} C_VEL
LIN {X 0,Y 56.577,Z 825.461,A -85,B 0,C 180,E1 4046.961,E2 4046.961} C_VEL
LIN {X 0,Y 58.411,Z 824.874,A -85,B 0,C 180,E1 4031.021,E2 4031.021} C_VEL
LIN {X 0,Y 65.735,Z 822.787,A -85,B 0,C 180,E1 4012.526,E2 4012.526} C_VEL
LIN {X 0,Y 77.861,Z 819.094,A -85,B 0,C 180,E1 3998.435,E2 3998.435} C_VEL
LIN {X 0,Y 93.153,Z 813.577,A -85,B 0,C 180,E1 3988.343,E2 3988.343} C_VEL
LIN {X 0,Y 109.626,Z 806.586,A -85,B 0,C 180,E1 3981.398,E2 3981.398} C_VEL
LIN {X 0,Y 127.092,Z 797.862,A -85,B 0,C 180,E1 3976.307,E2 3976.307} C_VEL
LIN {X 0,Y 144.447,Z 787.686,A -85,B 0,C 180,E1 3972.586,E2 3972.586} C_VEL
LIN {X 0,Y 161.325,Z 775.997,A -85,B 0,C 180,E1 3969.795,E2 3969.795} C_VEL
LIN {X 0,Y 177.545,Z 762.949,A -85,B 0,C 180,E1 3967.637,E2 3967.637} C_VEL
LIN {X 0,Y 193.487,Z 748.049,A -85,B 0,C 180,E1 3965.884,E2 3965.884} C_VEL
LIN {X 0,Y 207.964,Z 732.311,A -85,B 0,C 180,E1 3964.538,E2 3964.538} C_VEL
LIN {X 0,Y 221.363,Z 715.162,A -85,B 0,C 180,E1 3963.448,E2 3963.448} C_VEL
LIN {X 0,Y 233.199,Z 697.294,A -85,B 0,C 180,E1 3962.591,E2 3962.591} C_VEL
LIN {X 0,Y 239.133,Z 687.083,A -85,B 0,C 180,E1 3962.181,E2 3962.181} C_VEL
LIN {X 0,Y 228.04,Z 705.562,A -85,B 0,C 180,E1 3961.503,E2 3961.503} C_VEL
LIN {X 0,Y 215.477,Z 723.271,A -85,B 0,C 180,E1 3960.642,E2 3960.642} C_VEL
LIN {X 0,Y 201.472,Z 740.034,A -85,B 0,C 180,E1 3959.532,E2 3959.532} C_VEL
LIN {X 0,Y 186.071,Z 755.906,A -85,B 0,C 180,E1 3958.097,E2 3958.097} C_VEL
LIN {X 0,Y 170.161,Z 770.099,A -85,B 0,C 180,E1 3956.295,E2 3956.295} C_VEL
LIN {X 0,Y 152.849,Z 783.457,A -85,B 0,C 180,E1 3953.868,E2 3953.868} C_VEL
LIN {X 0,Y 134.79,Z 795.352,A -85,B 0,C 180,E1 3950.593,E2 3950.593} C_VEL
LIN {X 0,Y 117.31,Z 805.276,A -85,B 0,C 180,E1 3946.316,E2 3946.316} C_VEL
LIN {X 0,Y 99.008,Z 814.237,A -85,B 0,C 180,E1 3939.911,E2 3939.911} C_VEL
LIN {X 0,Y 87.933,Z 819.011,A -85,B 0,C 180,E1 3934.371,E2 3934.371} C_VEL
LIN {X 0,Y 81.863,Z 821.234,A -85,B 0,C 180,E1 3931.45,E2 3931.45} C_VEL
LIN {X 0,Y 64.008,Z 826.001,A -85,B 0,C 180,E1 3923.114,E2 3923.114} C_VEL
LIN {X 0,Y 59.575,Z 827.164,A -85,B 0,C 180,E1 3918.621,E2 3918.621} C_VEL
LIN {X 0,Y 50.556,Z 830.123,A -85,B 0,C 180,E1 3898.336,E2 3898.336} C_VEL
LIN {X 0,Y 48.307,Z 831.221,A -85,B 0,C 180,E1 3878.33,E2 3878.33} C_VEL
LIN {X 0,Y 48.45,Z 831.389,A -85,B 0,C 180,E1 3868.818,E2 3868.818} C_VEL
LIN {X 0,Y 48.765,Z 830.83,A -85,B 0,C 180,E1 3852.089,E2 3852.089} C_VEL
LIN {X 0,Y 54.137,Z 828.857,A -85,B 0,C 180,E1 3831.102,E2 3831.102} C_VEL
LIN {X 0,Y 66.06,Z 825.041,A -85,B 0,C 180,E1 3813.651,E2 3813.651} C_VEL
LIN {X 0,Y 81.938,Z 819.523,A -85,B 0,C 180,E1 3801.97,E2 3801.97} C_VEL
LIN {X 0,Y 100.027,Z 812.182,A -85,B 0,C 180,E1 3794.169,E2 3794.169} C_VEL
LIN {X 0,Y 119.375,Z 802.775,A -85,B 0,C 180,E1 3788.768,E2 3788.768} C_VEL
LIN {X 0,Y 137.546,Z 792.359,A -85,B 0,C 180,E1 3785.214,E2 3785.214} C_VEL
LIN {X 0,Y 156.122,Z 779.92,A -85,B 0,C 180,E1 3782.498,E2 3782.498} C_VEL
LIN {X 0,Y 172.979,Z 766.79,A -85,B 0,C 180,E1 3780.579,E2 3780.579} C_VEL
LIN {X 0,Y 189.059,Z 752.245,A -85,B 0,C 180,E1 3779.09,E2 3779.09} C_VEL
LIN {X 0,Y 204.098,Z 736.367,A -85,B 0,C 180,E1 3777.936,E2 3777.936} C_VEL
LIN {X 0,Y 208.14,Z 731.708,A -85,B 0,C 180,E1 3777.645,E2 3777.645} C_VEL
LIN {X 0,Y 193.828,Z 747.26,A -85,B 0,C 180,E1 3776.505,E2 3776.505} C_VEL
LIN {X 0,Y 177.651,Z 762.352,A -85,B 0,C 180,E1 3774.981,E2 3774.981} C_VEL
LIN {X 0,Y 161.14,Z 775.57,A -85,B 0,C 180,E1 3773.098,E2 3773.098} C_VEL
LIN {X 0,Y 143.883,Z 787.344,A -85,B 0,C 180,E1 3770.66,E2 3770.66} C_VEL
LIN {X 0,Y 126.02,Z 797.664,A -85,B 0,C 180,E1 3767.387,E2 3767.387} C_VEL
LIN {X 0,Y 107.056,Z 806.882,A -85,B 0,C 180,E1 3762.609,E2 3762.609} C_VEL
LIN {X 0,Y 89.628,Z 813.938,A -85,B 0,C 180,E1 3756.169,E2 3756.169} C_VEL
LIN {X 0,Y 73.139,Z 819.473,A -85,B 0,C 180,E1 3746.5,E2 3746.5} C_VEL
LIN {X 0,Y 59.557,Z 823.186,A -85,B 0,C 180,E1 3732.184,E2 3732.184} C_VEL
LIN {X 0,Y 50.895,Z 825.303,A -85,B 0,C 180,E1 3711.916,E2 3711.916} C_VEL
LIN {X 0,Y 48.604,Z 825.902,A -85,B 0,C 180,E1 3693.538,E2 3693.538} C_VEL
LIN {X 0,Y 49.416,Z 825.738,A -85,B 0,C 180,E1 3675.948,E2 3675.948} C_VEL
LIN {X 0,Y 55.522,Z 824.214,A -85,B 0,C 180,E1 3654.813,E2 3654.813} C_VEL
LIN {X 0,Y 68.162,Z 820.919,A -85,B 0,C 180,E1 3637.618,E2 3637.618} C_VEL
LIN {X 0,Y 83.856,Z 816.07,A -85,B 0,C 180,E1 3626.59,E2 3626.59} C_VEL
LIN {X 0,Y 101.559,Z 809.406,A -85,B 0,C 180,E1 3619.074,E2 3619.074} C_VEL
LIN {X 0,Y 119.524,Z 801.153,A -85,B 0,C 180,E1 3613.987,E2 3613.987} C_VEL
LIN {X 0,Y 137.221,Z 791.522,A -85,B 0,C 180,E1 3610.375,E2 3610.375} C_VEL
LIN {X 0,Y 154.369,Z 780.594,A -85,B 0,C 180,E1 3607.709,E2 3607.709} C_VEL
LIN {X 0,Y 171.782,Z 767.563,A -85,B 0,C 180,E1 3605.571,E2 3605.571} C_VEL
LIN {X 0,Y 187.638,Z 753.596,A -85,B 0,C 180,E1 3603.973,E2 3603.973} C_VEL
LIN {X 0,Y 202.69,Z 738.197,A -85,B 0,C 180,E1 3602.696,E2 3602.696} C_VEL
LIN {X 0,Y 207.726,Z 732.556,A -85,B 0,C 180,E1 3602.302,E2 3602.302} C_VEL
LIN {X 0,Y 193.011,Z 748.536,A -85,B 0,C 180,E1 3601.223,E2 3601.223} C_VEL
LIN {X 0,Y 176.971,Z 763.566,A -85,B 0,C 180,E1 3599.81,E2 3599.81} C_VEL
LIN {X 0,Y 160.072,Z 777.228,A -85,B 0,C 180,E1 3597.983,E2 3597.983} C_VEL
LIN {X 0,Y 142.403,Z 789.519,A -85,B 0,C 180,E1 3595.561,E2 3595.561} C_VEL
LIN {X 0,Y 124.11,Z 800.335,A -85,B 0,C 180,E1 3592.26,E2 3592.26} C_VEL
LIN {X 0,Y 105.456,Z 809.751,A -85,B 0,C 180,E1 3587.567,E2 3587.567} C_VEL
LIN {X 0,Y 86.934,Z 817.675,A -85,B 0,C 180,E1 3580.576,E2 3580.576} C_VEL
LIN {X 0,Y 70.149,Z 823.799,A -85,B 0,C 180,E1 3570.077,E2 3570.077} C_VEL
LIN {X 0,Y 59.575,Z 827.164,A -85,B 0,C 180,E1 3558.621,E2 3558.621} C_VEL
LIN {X 0,Y 54.8,Z 828.431,A -85,B 0,C 180,E1 3552.599,E2 3552.599} C_VEL
LIN {X 0,Y 44.362,Z 830.069,A -85,B 0,C 180,E1 3538.21,E2 3538.21} C_VEL
LIN {X 0,Y 40.681,Z 830.628,A -85,B 0,C 180,E1 3526.363,E2 3526.363} C_VEL
LIN {X 0,Y 40.409,Z 830.695,A -85,B 0,C 180,E1 3523.224,E2 3523.224} C_VEL
LIN {X 0,Y 40.485,Z 830.961,A -85,B 0,C 180,E1 3510,E2 3510} C_VEL
LIN {X 0,Y 40.773,Z 830.532,A -85,B 0,C 180,E1 3491.411,E2 3491.411} C_VEL
LIN {X 0,Y 47.478,Z 828.524,A -85,B 0,C 180,E1 3465.978,E2 3465.978} C_VEL
LIN {X 0,Y 61.089,Z 824.798,A -85,B 0,C 180,E1 3447.896,E2 3447.896} C_VEL
LIN {X 0,Y 78.324,Z 819.375,A -85,B 0,C 180,E1 3436.785,E2 3436.785} C_VEL
LIN {X 0,Y 97.383,Z 812.094,A -85,B 0,C 180,E1 3429.723,E2 3429.723} C_VEL
LIN {X 0,Y 116.452,Z 803.257,A -85,B 0,C 180,E1 3425.156,E2 3425.156} C_VEL
LIN {X 0,Y 135.062,Z 793.064,A -85,B 0,C 180,E1 3422.031,E2 3422.031} C_VEL
LIN {X 0,Y 152.975,Z 781.585,A -85,B 0,C 180,E1 3419.78,E2 3419.78} C_VEL
LIN {X 0,Y 171.346,Z 767.768,A -85,B 0,C 180,E1 3417.993,E2 3417.993} C_VEL
LIN {X 0,Y 176.65,Z 763.248,A -85,B 0,C 180,E1 3417.547,E2 3417.547} C_VEL
LIN {X 0,Y 159.389,Z 776.735,A -85,B 0,C 180,E1 3415.858,E2 3415.858} C_VEL
LIN {X 0,Y 141.824,Z 788.435,A -85,B 0,C 180,E1 3413.73,E2 3413.73} C_VEL
LIN {X 0,Y 123.55,Z 798.629,A -85,B 0,C 180,E1 3410.854,E2 3410.854} C_VEL
LIN {X 0,Y 104.752,Z 807.41,A -85,B 0,C 180,E1 3406.796,E2 3406.796} C_VEL
LIN {X 0,Y 85.789,Z 814.685,A -85,B 0,C 180,E1 3400.737,E2 3400.737} C_VEL
LIN {X 0,Y 68.204,Z 820.133,A -85,B 0,C 180,E1 3391.59,E2 3391.59} C_VEL
LIN {X 0,Y 52.603,Z 823.94,A -85,B 0,C 180,E1 3376.243,E2 3376.243} C_VEL
LIN {X 0,Y 43.22,Z 825.815,A -85,B 0,C 180,E1 3354.607,E2 3354.607} C_VEL
LIN {X 0,Y 40.582,Z 826.393,A -85,B 0,C 180,E1 3331.412,E2 3331.412} C_VEL
LIN {X 0,Y 42.357,Z 826.022,A -85,B 0,C 180,E1 3309.264,E2 3309.264} C_VEL
LIN {X 0,Y 50.235,Z 824.457,A -85,B 0,C 180,E1 3287.414,E2 3287.414} C_VEL
LIN {X 0,Y 64.296,Z 821.178,A -85,B 0,C 180,E1 3271.21,E2 3271.21} C_VEL
LIN {X 0,Y 81.411,Z 816.235,A -85,B 0,C 180,E1 3261.032,E2 3261.032} C_VEL
LIN {X 0,Y 100.12,Z 809.501,A -85,B 0,C 180,E1 3254.379,E2 3254.379} C_VEL
LIN {X 0,Y 118.775,Z 801.167,A -85,B 0,C 180,E1 3249.972,E2 3249.972} C_VEL
LIN {X 0,Y 136.962,Z 791.427,A -85,B 0,C 180,E1 3246.875,E2 3246.875} C_VEL
LIN {X 0,Y 155.452,Z 779.693,A -85,B 0,C 180,E1 3244.495,E2 3244.495} C_VEL
LIN {X 0,Y 172.175,Z 767.249,A -85,B 0,C 180,E1 3242.793,E2 3242.793} C_VEL
LIN {X 0,Y 176.125,Z 763.93,A -85,B 0,C 180,E1 3242.401,E2 3242.401} C_VEL
LIN {X 0,Y 157.789,Z 778.326,A -85,B 0,C 180,E1 3240.727,E2 3240.727} C_VEL
LIN {X 0,Y 140.015,Z 790.258,A -85,B 0,C 180,E1 3238.646,E2 3238.646} C_VEL
LIN {X 0,Y 120.339,Z 801.456,A -85,B 0,C 180,E1 3235.573,E2 3235.573} C_VEL
LIN {X 0,Y 101.142,Z 810.553,A -85,B 0,C 180,E1 3231.319,E2 3231.319} C_VEL
LIN {X 0,Y 82.739,Z 817.849,A -85,B 0,C 180,E1 3225.18,E2 3225.18} C_VEL
LIN {X 0,Y 64.955,Z 823.739,A -85,B 0,C 180,E1 3215.253,E2 3215.253} C_VEL
LIN {X 0,Y 49.96,Z 827.959,A -85,B 0,C 180,E1 3198.67,E2 3198.67} C_VEL
LIN {X 0,Y 41.713,Z 830.15,A -85,B 0,C 180,E1 3175.56,E2 3175.56} C_VEL
LIN {X 0,Y 40.409,Z 830.695,A -85,B 0,C 180,E1 3163.224,E2 3163.224} C_VEL
LIN {X 0,Y 39.442,Z 830.856,A -85,B 0,C 180,E1 3154.673,E2 3154.673} C_VEL
LIN {X 0,Y 37.322,Z 830.702,A -85,B 0,C 180,E1 3143.455,E2 3143.455} C_VEL
LIN {X 0,Y 35.822,Z 829.511,A -85,B 0,C 180,E1 3114.342,E2 3114.342} C_VEL
LIN {X 0,Y 37.299,Z 829.113,A -85,B 0,C 180,E1 3108.454,E2 3108.454} C_VEL
LIN {X 0,Y 51.193,Z 825.966,A -85,B 0,C 180,E1 3086.051,E2 3086.051} C_VEL
LIN {X 0,Y 69.014,Z 821.16,A -85,B 0,C 180,E1 3073.915,E2 3073.915} C_VEL
LIN {X 0,Y 88.606,Z 814.594,A -85,B 0,C 180,E1 3066.786,E2 3066.786} C_VEL
LIN {X 0,Y 108.077,Z 806.584,A -85,B 0,C 180,E1 3062.408,E2 3062.408} C_VEL
LIN {X 0,Y 127.986,Z 796.583,A -85,B 0,C 180,E1 3059.354,E2 3059.354} C_VEL
LIN {X 0,Y 144.937,Z 786.54,A -85,B 0,C 180,E1 3057.406,E2 3057.406} C_VEL
LIN {X 0,Y 125.452,Z 797.588,A -85,B 0,C 180,E1 3055.023,E2 3055.023} C_VEL
LIN {X 0,Y 106.075,Z 806.691,A -85,B 0,C 180,E1 3051.768,E2 3051.768} C_VEL
LIN {X 0,Y 87.166,Z 813.962,A -85,B 0,C 180,E1 3047.157,E2 3047.157} C_VEL
LIN {X 0,Y 68.192,Z 819.662,A -85,B 0,C 180,E1 3039.778,E2 3039.778} C_VEL
LIN {X 0,Y 51.006,Z 823.645,A -85,B 0,C 180,E1 3027.447,E2 3027.447} C_VEL
LIN {X 0,Y 37.797,Z 826.022,A -85,B 0,C 180,E1 3005.588,E2 3005.588} C_VEL
LIN {X 0,Y 32.82,Z 826.759,A -85,B 0,C 180,E1 2978.761,E2 2978.761} C_VEL
LIN {X 0,Y 33.057,Z 826.728,A -85,B 0,C 180,E1 2957.777,E2 2957.777} C_VEL
LIN {X 0,Y 39.808,Z 825.749,A -85,B 0,C 180,E1 2929.23,E2 2929.23} C_VEL
LIN {X 0,Y 54.039,Z 823.099,A -85,B 0,C 180,E1 2909.588,E2 2909.588} C_VEL
LIN {X 0,Y 71.677,Z 818.769,A -85,B 0,C 180,E1 2898.462,E2 2898.462} C_VEL
LIN {X 0,Y 91.809,Z 812.365,A -85,B 0,C 180,E1 2891.443,E2 2891.443} C_VEL
LIN {X 0,Y 110.866,Z 804.752,A -85,B 0,C 180,E1 2887.242,E2 2887.242} C_VEL
LIN {X 0,Y 130.334,Z 795.226,A -85,B 0,C 180,E1 2884.239,E2 2884.239} C_VEL
LIN {X 0,Y 144.707,Z 786.866,A -85,B 0,C 180,E1 2882.524,E2 2882.524} C_VEL
LIN {X 0,Y 124.98,Z 798.324,A -85,B 0,C 180,E1 2880.243,E2 2880.243} C_VEL
LIN {X 0,Y 105.123,Z 807.969,A -85,B 0,C 180,E1 2877.031,E2 2877.031} C_VEL
LIN {X 0,Y 85.743,Z 815.779,A -85,B 0,C 180,E1 2872.38,E2 2872.38} C_VEL
LIN {X 0,Y 65.441,Z 822.312,A -85,B 0,C 180,E1 2864.265,E2 2864.265} C_VEL
LIN {X 0,Y 48.146,Z 826.712,A -85,B 0,C 180,E1 2850.715,E2 2850.715} C_VEL
LIN {X 0,Y 35.629,Z 829.449,A -85,B 0,C 180,E1 2826.108,E2 2826.108} C_VEL
LIN {X 0,Y 32.337,Z 830.409,A -85,B 0,C 180,E1 2797.104,E2 2797.104} C_VEL
LIN {X 0,Y 32.402,Z 830.462,A -85,B 0,C 180,E1 2786.462,E2 2786.462} C_VEL
LIN {X 0,Y 34.516,Z 829.672,A -85,B 0,C 180,E1 2758.573,E2 2758.573} C_VEL
LIN {X 0,Y 37.299,Z 829.113,A -85,B 0,C 180,E1 2748.454,E2 2748.454} C_VEL
LIN {X 0,Y 40.626,Z 828.199,A -85,B 0,C 180,E1 2738.208,E2 2738.208} C_VEL
LIN {X 0,Y 52.04,Z 824.75,A -85,B 0,C 180,E1 2715.257,E2 2715.257} C_VEL
LIN {X 0,Y 56.945,Z 823.468,A -85,B 0,C 180,E1 2711.617,E2 2711.617} C_VEL
LIN {X 0,Y 78.426,Z 817.387,A -85,B 0,C 180,E1 2703.653,E2 2703.653} C_VEL
LIN {X 0,Y 98.989,Z 809.921,A -85,B 0,C 180,E1 2699.354,E2 2699.354} C_VEL
LIN {X 0,Y 113.109,Z 803.735,A -85,B 0,C 180,E1 2697.276,E2 2697.276} C_VEL
LIN {X 0,Y 92.506,Z 812.033,A -85,B 0,C 180,E1 2693.914,E2 2693.914} C_VEL
LIN {X 0,Y 72.373,Z 818.418,A -85,B 0,C 180,E1 2688.773,E2 2688.773} C_VEL
LIN {X 0,Y 52.294,Z 823.192,A -85,B 0,C 180,E1 2679.529,E2 2679.529} C_VEL
LIN {X 0,Y 35.487,Z 825.954,A -85,B 0,C 180,E1 2662.082,E2 2662.082} C_VEL
LIN {X 0,Y 25.523,Z 827.151,A -85,B 0,C 180,E1 2628.264,E2 2628.264} C_VEL
LIN {X 0,Y 24.807,Z 827.235,A -85,B 0,C 180,E1 2600.722,E2 2600.722} C_VEL
LIN {X 0,Y 30.421,Z 826.618,A -85,B 0,C 180,E1 2568.904,E2 2568.904} C_VEL
LIN {X 0,Y 46.287,Z 824.302,A -85,B 0,C 180,E1 2544.874,E2 2544.874} C_VEL
LIN {X 0,Y 64.885,Z 820.44,A -85,B 0,C 180,E1 2533.886,E2 2533.886} C_VEL
LIN {X 0,Y 85.713,Z 814.517,A -85,B 0,C 180,E1 2527.472,E2 2527.472} C_VEL
LIN {X 0,Y 106.195,Z 806.878,A -85,B 0,C 180,E1 2523.63,E2 2523.63} C_VEL
LIN {X 0,Y 112.725,Z 804.047,A -85,B 0,C 180,E1 2522.629,E2 2522.629} C_VEL
LIN {X 0,Y 91.894,Z 812.773,A -85,B 0,C 180,E1 2519.378,E2 2519.378} C_VEL
LIN {X 0,Y 71.345,Z 819.676,A -85,B 0,C 180,E1 2514.263,E2 2514.263} C_VEL
LIN {X 0,Y 51.677,Z 824.815,A -85,B 0,C 180,E1 2505.325,E2 2505.325} C_VEL
LIN {X 0,Y 34.478,Z 828.145,A -85,B 0,C 180,E1 2487.243,E2 2487.243} C_VEL
LIN {X 0,Y 24.83,Z 829.792,A -85,B 0,C 180,E1 2451.248,E2 2451.248} C_VEL
LIN {X 0,Y 24.485,Z 830.063,A -85,B 0,C 180,E1 2430,E2 2430} C_VEL
LIN {X 0,Y 26.562,Z 829.456,A -85,B 0,C 180,E1 2395.625,E2 2395.625} C_VEL
LIN {X 0,Y 38.959,Z 827.341,A -85,B 0,C 180,E1 2366.073,E2 2366.073} C_VEL
LIN {X 0,Y 56.945,Z 823.468,A -85,B 0,C 180,E1 2351.617,E2 2351.617} C_VEL
LIN {X 0,Y 61.019,Z 822.395,A -85,B 0,C 180,E1 2348.599,E2 2348.599} C_VEL
LIN {X 0,Y 70.821,Z 819.299,A -85,B 0,C 180,E1 2339.705,E2 2339.705} C_VEL
LIN {X 0,Y 74.722,Z 818.061,A -85,B 0,C 180,E1 2338.245,E2 2338.245} C_VEL
LIN {X 0,Y 80.589,Z 816.203,A -85,B 0,C 180,E1 2337.108,E2 2337.108} C_VEL
LIN {X 0,Y 60.538,Z 821.497,A -85,B 0,C 180,E1 2332.285,E2 2332.285} C_VEL
LIN {X 0,Y 39.881,Z 825.304,A -85,B 0,C 180,E1 2322.301,E2 2322.301} C_VEL
LIN {X 0,Y 22.861,Z 827.23,A -85,B 0,C 180,E1 2298.029,E2 2298.029} C_VEL
LIN {X 0,Y 16.633,Z 827.738,A -85,B 0,C 180,E1 2253.446,E2 2253.446} C_VEL
LIN {X 0,Y 21.576,Z 827.374,A -85,B 0,C 180,E1 2205.965,E2 2205.965} C_VEL
LIN {X 0,Y 37.185,Z 825.712,A -85,B 0,C 180,E1 2179.765,E2 2179.765} C_VEL
LIN {X 0,Y 56.679,Z 822.347,A -85,B 0,C 180,E1 2168.94,E2 2168.94} C_VEL
LIN {X 0,Y 78.114,Z 817.021,A -85,B 0,C 180,E1 2163.277,E2 2163.277} C_VEL
LIN {X 0,Y 80.306,Z 816.378,A -85,B 0,C 180,E1 2162.78,E2 2162.78} C_VEL
LIN {X 0,Y 59.033,Z 822.344,A -85,B 0,C 180,E1 2157.815,E2 2157.815} C_VEL
LIN {X 0,Y 38.839,Z 826.485,A -85,B 0,C 180,E1 2148.021,E2 2148.021} C_VEL
LIN {X 0,Y 22.242,Z 828.773,A -85,B 0,C 180,E1 2124.011,E2 2124.011} C_VEL
LIN {X 0,Y 16.407,Z 829.595,A -85,B 0,C 180,E1 2073.494,E2 2073.494} C_VEL
LIN {X 0,Y 16.904,Z 829.397,A -85,B 0,C 180,E1 2045.542,E2 2045.542} C_VEL
LIN {X 0,Y 29.117,Z 827.906,A -85,B 0,C 180,E1 2002.005,E2 2002.005} C_VEL
LIN {X 0,Y 48.288,Z 824.684,A -85,B 0,C 180,E1 1986.349,E2 1986.349} C_VEL
LIN {X 0,Y 68.991,Z 819.683,A -85,B 0,C 180,E1 1979.481,E2 1979.481} C_VEL
LIN {X 0,Y 74.722,Z 818.061,A -85,B 0,C 180,E1 1978.245,E2 1978.245} C_VEL
LIN {X 0,Y 73.14,Z 818.493,A -85,B 0,C 180,E1 1977.504,E2 1977.504} C_VEL
LIN {X 0,Y 64.467,Z 820.695,A -85,B 0,C 180,E1 1976.879,E2 1976.879} C_VEL
LIN {X 0,Y 45.973,Z 824.681,A -85,B 0,C 180,E1 1977.952,E2 1977.952} C_VEL
LIN {X 0,Y 34.967,Z 826.418,A -85,B 0,C 180,E1 1980.963,E2 1980.963} C_VEL
LIN {X 0,Y 15.993,Z 828.537,A -85,B 0,C 180,E1 2000.32,E2 2000.32} C_VEL
LIN {X 0,Y 8.447,Z 829.163,A -85,B 0,C 180,E1 2070,E2 2070} C_VEL
LIN {X 0,Y 18.643,Z 828.314,A -85,B 0,C 180,E1 2144.869,E2 2144.869} C_VEL
LIN {X 0,Y 38.996,Z 825.846,A -85,B 0,C 180,E1 2160.708,E2 2160.708} C_VEL
LIN {X 0,Y 46.349,Z 824.568,A -85,B 0,C 180,E1 2163.07,E2 2163.07} C_VEL
LIN {X 0,Y 25.727,Z 827.21,A -85,B 0,C 180,E1 2173.691,E2 2173.691} C_VEL
LIN {X 0,Y 10.843,Z 828.076,A -85,B 0,C 180,E1 2209.797,E2 2209.797} C_VEL
LIN {X 0,Y 9.388,Z 828.125,A -85,B 0,C 180,E1 2275.215,E2 2275.215} C_VEL
LIN {X 0,Y 22.04,Z 827.439,A -85,B 0,C 180,E1 2322.297,E2 2322.297} C_VEL
LIN {X 0,Y 42.125,Z 825.159,A -85,B 0,C 180,E1 2335.453,E2 2335.453} C_VEL
LIN {X 0,Y 46.46,Z 824.5,A -85,B 0,C 180,E1 2336.895,E2 2336.895} C_VEL
LIN {X 0,Y 34.967,Z 826.418,A -85,B 0,C 180,E1 2340.963,E2 2340.963} C_VEL
LIN {X 0,Y 27.048,Z 827.4,A -85,B 0,C 180,E1 2343.471,E2 2343.471} C_VEL
LIN {X 0,Y 14.849,Z 828.293,A -85,B 0,C 180,E1 2342.955,E2 2342.955} C_VEL
LIN {X 0,Y 0.985,Z 828.657,A -85,B 0,C 180,E1 2301.608,E2 2301.608} C_VEL
LIN {X 0,Y 2.242,Z 828.618,A -85,B 0,C 180,E1 2174.882,E2 2174.882} C_VEL
LIN {X 0,Y 4.487,Z 828.576,A -85,B 0,C 180,E1 2165.08,E2 2165.08} C_VEL
LIN {X 0,Y 0.373,Z 828.71,A -85,B 0,C 180,E1 2069.999,E2 2069.999} C_VEL
LIN {X 0,Y 4.707,Z 828.562,A -85,B 0,C 180,E1 1974.655,E2 1974.655} C_VEL
LIN {X 0,Y 2.242,Z 828.618,A -85,B 0,C 180,E1 1814.882,E2 1814.882} C_VEL
LIN {X 0,Y 4.233,Z 830.617,A -85,B 0,C 180,E1 1806.588,E2 1806.588} C_VEL
LIN {X 0,Y 4.233,Z 862.5,A -85,B 0,C 180,E1 1806.588,E2 1806.588} C_VEL
LIN {X 0,Y 4.233,Z 862.5,A -85,B 0,C 180,E1 1806.588,E2 1806.588}

QRS_NEXT_CUT()

QRS_NEXT()
QRS_HOME()

END
